PROGRAM MAIN
VAR
    stJointBench : ST_JointBenchAds := (
        sDeviceName := 'Ti5 Harmonic Joint',
        nVendorId := 0,
        nProductCode := 0,
        nRevision := 0
    );
    fbJointBenchAxis : FB_JointBenchAxis;
END_VAR


fbJointBenchAxis(stIf := stJointBench);

END_PROGRAM

(* stored: Version 1.1.0.1, ProductVersion 3.1.4024.0
   POU MAIN: PouType Program *)
